KUKA KRL program: SetPlacePos_P1L1.src, SetPlacePos_P1L1.dat

--- SetPlacePos_P1L1.src ---
&ACCESS RVO1
&PARAM EDITMASK = *
DEF SetPlacePos_P1L1()
   ;Esses valores devem vir sempre da main

   ;XPlace     = faz o place no devido local
   XApp1Place = MatrizPontos[MosaicoAtivo,PlaceAtivo+1].XApp1Place
   XApp2Place = MatrizPontos[MosaicoAtivo,PlaceAtivo+1].XApp2Place
   XPlace     = MatrizPontos[MosaicoAtivo,PlaceAtivo+1].XPlace

   ;CamadaAtiva
   XApp1Place.Z = XApp1Place.Z + (CamadaAtiva)*AlturaCaixa
   XApp2Place.Z = XApp2Place.Z + (CamadaAtiva)*AlturaCaixa
   XPlace.Z=XPlace.Z + (CamadaAtiva)*AlturaCaixa
END

--- SetPlacePos_P1L1.dat ---
DEFDAT SetPlacePos_P1L1
ENDDAT
